PROGRAM MAIN
VAR
END_VAR

END_PROGRAM

(* stored: Version 1.1.0.1
   POU MAIN: Id {7dbc7edd-3617-4d47-b497-c178be1f499a} *)
